(* Schneider Machine Expert - Basic project _M5.4 Schedule Block, file version 2.6.0.0 *)
(* CompanyInformations: Name=Schneider Electric, PhoneNumber=+44 870 608 8608, Street=Stafford Park 5, City=Telford, ZipCode=TF3 3BL, Country=United Kingdom, WebSite=se.com/uk *)
(* ProjectInformations: Name=Training M221, Description=Training of the Modicon M221.
We are going to work with a Conveyor belt machine.
During this trainignn we will add more features to this machine to understand how to use the software. *)
(* UserInformations: LastName=Ahumada, FirstName=Leandro, PhoneNumber=+44 870 608 8608, CellNumber=+44 870 608 8608, Email=gb-customerservices@schneider-electric.com, Street=Stafford Park 5, City=Telford, ZipCode=TF3 3BL, Country=United Kingdom *)

HARDWARE
  Cpu 0: TM221CE24R
  EthernetConfiguration: NetworkName=M221, IpAllocationMode=FixedAddress, IpAddress=192.168.1.221, SubnetMask=255.255.255.0
  SerialLineConfiguration: Baud=Baud19200, Parity=ParityEven, DataBits=DataBits8, StopBits=StopBits1, PhysicalMedium=PhysicalMediumRs485, TransmissionMode=TransmissionModeModbusRtu, SlaveId=1, Addressing=SlaveAddressing
  MastTask: UsePeriodScanMode=false, PeriodScan=100
  FastTask: Period=255
  CpuBehavior: StartingMode=StartAsPreviousState, AutoSaveRamOnEeprom=true, WatchdogPeriod=250

SYMBOLS  (address, symbol, comment, settings)
  %M0       AUX_MOTOR  "Auxiliar motor"
  %M1       AUX_MACHINE  "Auxiliar Machine"
  %M10      MI_START  "M Start pushbutton"
  %M11      MI_STOP  "M Stop pushbutton"
  %M12      MI_SENSOR  "M Photo-Electric sensor"
  %M20      CMD_COUNTER_RESET
  %M21      IND_COUNTER_REACHED
  %M22      CFG_SCH_MONDAY
  %M23      CFG_SCH_TUESDAY
  %M24      CFG_SCH_WEDNESDAY
  %M25      CFG_SCH_THURSDAY
  %M26      CFG_SCH_FRIDAY
  %M27      CFG_SCH_SATURDAY
  %M28      CFG_SCH_SUNDAY
  %M80      PET_RTC_ENABLE  "At state 1, the RD and WR input values are read continuously to determine the action to take."
  %M81      PET_RTC_READ  "RD = 1 and WR = 0. Read the RTC value."
  %M82      PET_RTC_WRITE  "RD = 0 and WR = 1. When the rising edge of WR is detected, update the RTC using the object values specified in the RTC parameter"
  %M83      IND_RTC_DONE  "Set to 1 when the RTC is successfully read from or written to."
  %M84      IND_RTC_ERROR  "The ErrorId output object indicates the cause of the error."
  %M90      IND_ALARM_SYSTEM
  %M100     PET_ACK
  %M101     ALARM_01
  %M102     ALARM_02
  %MW0      IND_MOTOR_COUNTER
  %MW1      IND_MOTOR_TIME
  %MW2      AUX_RTC_ACTUAL_TOTAL_MM
  %MW3      AUX_MACHINE_ON_TOTAL_MM
  %MW4      AUX_MACHINE_OFF_TOTAL_MM
  %MW10     CFG_TIMER_MOTOR
  %MW11     CFG_COUNTER_MOTOR
  %MW12     CFG_MACHINE_ON_HH
  %MW13     CFG_MACHINE_ON_MM
  %MW14     CFG_MACHINE_OFF_HH
  %MW15     CFG_MACHINE_OFF_MM
  %MW20     CFG_SCH_STARTDAY  "Config. - Schedule - Start day"
  %MW21     CFG_SCH_STARTMONTH  "Config. - Schedule - Start month"
  %MW22     CFG_SCH_STARTHOUR  "Config. - Schedule - Start hour"
  %MW23     CFG_SCH_STARTMIN  "Config. - Schedule - Start min"
  %MW24     CFG_SCH_ENDDAY  "Config. - Schedule - End day"
  %MW25     CFG_SCH_ENDMONTH  "Config. - Schedule - End month"
  %MW26     CFG_SCH_ENDHOUR  "Config. - Schedule - End hour"
  %MW27     CFG_SCH_ENDMIN
  %MW28     CFG_SCH_DOW  "Config. - Schedule - Day of week"
  %MW41     IND_RTC_IDERROR
  %MW42     IND_RTC_ACTUAL_DAY
  %MW43     IND_RTC_ACTUAL_MONTH
  %MW44     IND_RTC_ACTUAL_YEAR
  %MW45     IND_RTC_ACTUAL_HH
  %MW46     IND_RTC_ACTUAL_MM
  %MW47     IND_RTC_ACTUAL_SS
  %MW48     IND_RTC_ACTUAL_DAYOFWEEK
  %MW50     IND_RTC_WRITE_DAY
  %MW51     IND_RTC_WRITE_MONTH
  %MW52     IND_RTC_WRITE_YEAR
  %MW53     IND_RTC_WRITE_HH
  %MW54     IND_RTC_WRITE_MM
  %MW55     IND_RTC_WRITE_SS
  %MW100    VAR_A
  %MW101    VAR_B
  %MW102    VAR_C
  %MF104    VAR_D
  %TM0      TIMER_MOTOR_ON  [Preset=5, Base=OneSecond]
  %SCH0       [Configured=true, OutputBit=%M1, StartDate=2012-01-01T00:00:00, EndDate=2012-01-01T00:00:00]
  %RTC0     INST_RTC  [Day(Value(int=24)), Month(Value(int=12)), Year(Value(int=2019)), Hours(Value(int=0)), Minutes(Value(int=0)), Seconds(Value(int=0))]
  %I0.0     I_START  "Start pushbutton"
  %I0.1     I_STOP  "Stop pushbutton"
  %I0.5     I_SENSOR  "Photo-Electric sensor"
  %Q0.0     Q_MOTOR  "Motor"
  %Q0.1     Q_MACHINE_ON
  %Q0.2     Q_ALARM
  %Q0.3     Q_MACHINE_DISABLED

POU PRG_CONFIG
  (* SectionNumber=1 *)

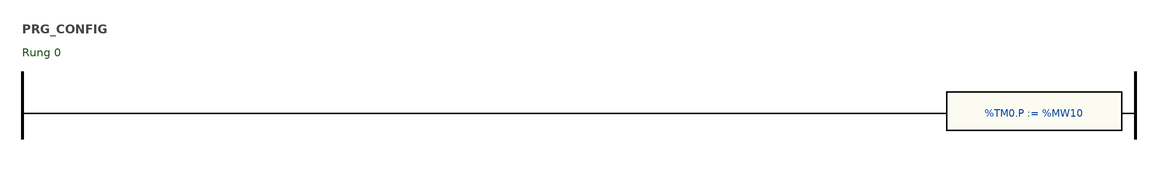

// Rung 0
  LD 1
  [ %TM0.P := %MW10 ]     (* TIMER_MOTOR_ON, CFG_TIMER_MOTOR *)
  // as ST:
  //   TIMER_MOTOR_ON.P := CFG_TIMER_MOTOR;

POU PRG_RTC
  (* SectionNumber=2 *)

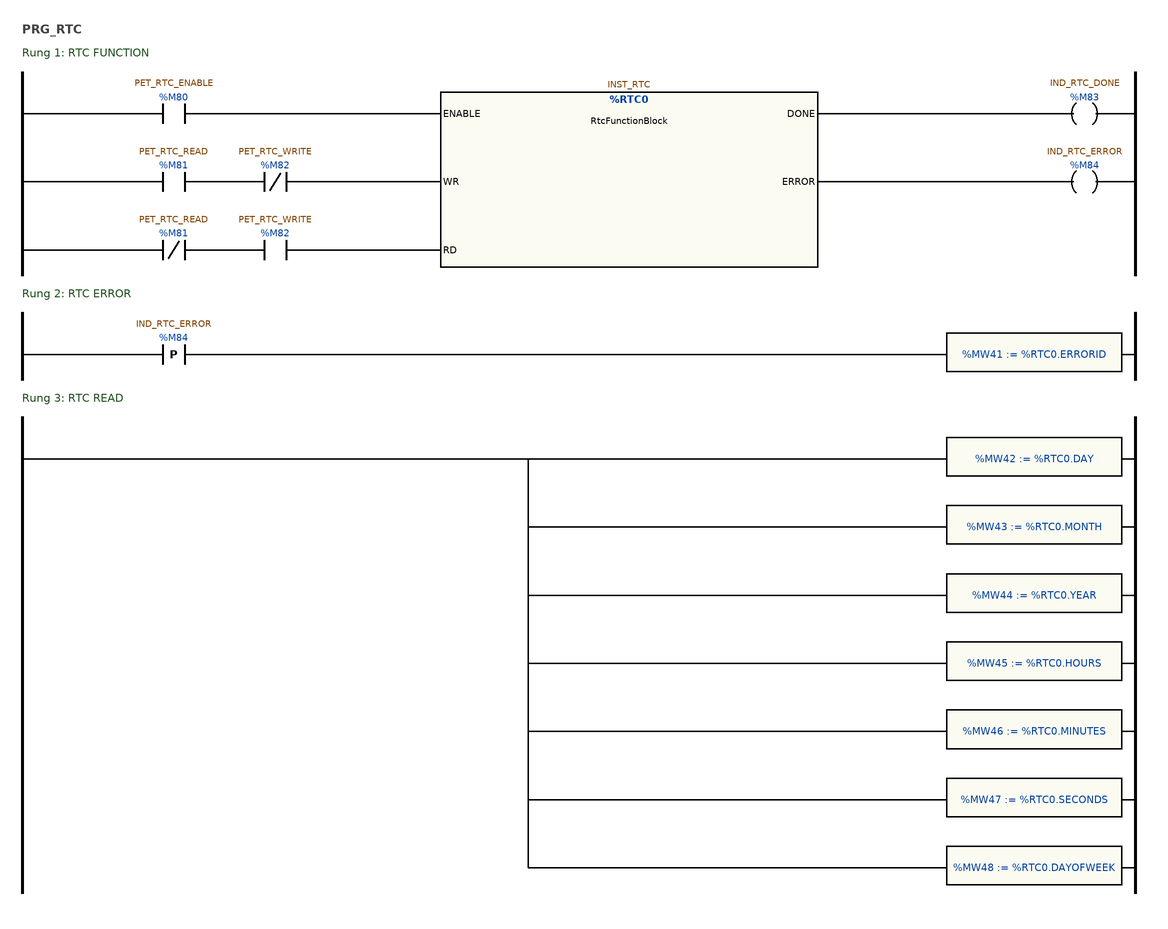

// Rung 1: RTC FUNCTION
  BLK %RTC0               (* INST_RTC *)
  LD %M80                 (* PET_RTC_ENABLE *)
  ENABLE
  LD %M81                 (* PET_RTC_READ *)
  ANDN %M82               (* PET_RTC_WRITE *)
  WR
  LDN %M81                (* PET_RTC_READ *)
  AND %M82                (* PET_RTC_WRITE *)
  RD
  OUT_BLK
  LD DONE
  ST %M83                 (* IND_RTC_DONE *)
  LD ERROR
  ST %M84                 (* IND_RTC_ERROR *)
  END_BLK
  // as ST:
  //   INST_RTC(ENABLE := PET_RTC_ENABLE, WR := PET_RTC_READ AND NOT PET_RTC_WRITE, RD := NOT PET_RTC_READ AND PET_RTC_WRITE);
  //   IND_RTC_DONE := INST_RTC.DONE;
  //   IND_RTC_ERROR := INST_RTC.ERROR;

// Rung 2: RTC ERROR
  LDR %M84                (* IND_RTC_ERROR *)
  [ %MW41 := %RTC0.ERRORID ](* IND_RTC_IDERROR, INST_RTC *)
  // as ST:
  //   IF RISING(IND_RTC_ERROR) THEN IND_RTC_IDERROR := INST_RTC.ERRORID; END_IF;

// Rung 3: RTC READ
  LD 1
  [ %MW42 := %RTC0.DAY ]  (* IND_RTC_ACTUAL_DAY, INST_RTC *)
  [ %MW43 := %RTC0.MONTH ](* IND_RTC_ACTUAL_MONTH, INST_RTC *)
  [ %MW44 := %RTC0.YEAR ] (* IND_RTC_ACTUAL_YEAR, INST_RTC *)
  [ %MW45 := %RTC0.HOURS ](* IND_RTC_ACTUAL_HH, INST_RTC *)
  [ %MW46 := %RTC0.MINUTES ](* IND_RTC_ACTUAL_MM, INST_RTC *)
  [ %MW47 := %RTC0.SECONDS ](* IND_RTC_ACTUAL_SS, INST_RTC *)
  [ %MW48 := %RTC0.DAYOFWEEK ](* IND_RTC_ACTUAL_DAYOFWEEK, INST_RTC *)
  // as ST:
  //   IND_RTC_ACTUAL_DAY := INST_RTC.DAY;
  //   IND_RTC_ACTUAL_MONTH := INST_RTC.MONTH;
  //   IND_RTC_ACTUAL_YEAR := INST_RTC.YEAR;
  //   IND_RTC_ACTUAL_HH := INST_RTC.HOURS;
  //   IND_RTC_ACTUAL_MM := INST_RTC.MINUTES;
  //   IND_RTC_ACTUAL_SS := INST_RTC.SECONDS;
  //   IND_RTC_ACTUAL_DAYOFWEEK := INST_RTC.DAYOFWEEK;

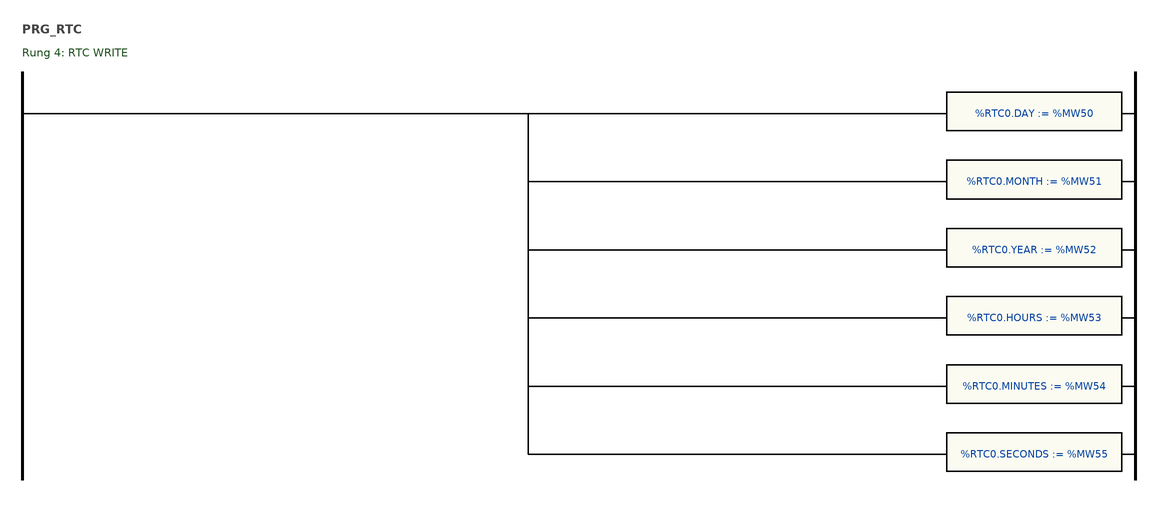

// Rung 4: RTC WRITE
  LD 1
  [ %RTC0.DAY := %MW50 ]  (* INST_RTC, IND_RTC_WRITE_DAY *)
  [ %RTC0.MONTH := %MW51 ](* INST_RTC, IND_RTC_WRITE_MONTH *)
  [ %RTC0.YEAR := %MW52 ] (* INST_RTC, IND_RTC_WRITE_YEAR *)
  [ %RTC0.HOURS := %MW53 ](* INST_RTC, IND_RTC_WRITE_HH *)
  [ %RTC0.MINUTES := %MW54 ](* INST_RTC, IND_RTC_WRITE_MM *)
  [ %RTC0.SECONDS := %MW55 ](* INST_RTC, IND_RTC_WRITE_SS *)
  // as ST:
  //   INST_RTC.DAY := IND_RTC_WRITE_DAY;
  //   INST_RTC.MONTH := IND_RTC_WRITE_MONTH;
  //   INST_RTC.YEAR := IND_RTC_WRITE_YEAR;
  //   INST_RTC.HOURS := IND_RTC_WRITE_HH;
  //   INST_RTC.MINUTES := IND_RTC_WRITE_MM;
  //   INST_RTC.SECONDS := IND_RTC_WRITE_SS;

POU PRG_SCHEDULE
  (* SectionNumber=3 *)

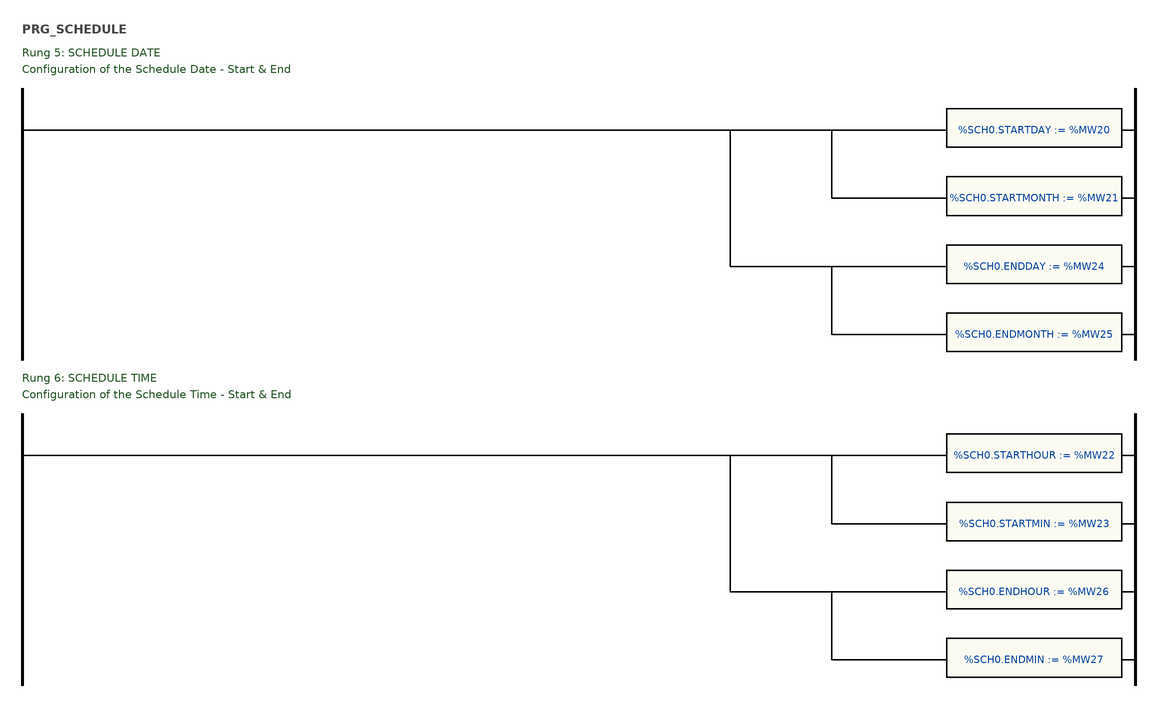

// Rung 5: SCHEDULE DATE
// Configuration of the Schedule Date - Start & End
  LD 1
  [ %SCH0.STARTDAY := %MW20 ](* CFG_SCH_STARTDAY *)
  [ %SCH0.STARTMONTH := %MW21 ](* CFG_SCH_STARTMONTH *)
  [ %SCH0.ENDDAY := %MW24 ](* CFG_SCH_ENDDAY *)
  [ %SCH0.ENDMONTH := %MW25 ](* CFG_SCH_ENDMONTH *)
  // as ST:
  //   %SCH0.STARTDAY := CFG_SCH_STARTDAY;
  //   %SCH0.STARTMONTH := CFG_SCH_STARTMONTH;
  //   %SCH0.ENDDAY := CFG_SCH_ENDDAY;
  //   %SCH0.ENDMONTH := CFG_SCH_ENDMONTH;

// Rung 6: SCHEDULE TIME
// Configuration of the Schedule Time - Start & End
  LD 1
  [ %SCH0.STARTHOUR := %MW22 ](* CFG_SCH_STARTHOUR *)
  [ %SCH0.STARTMIN := %MW23 ](* CFG_SCH_STARTMIN *)
  [ %SCH0.ENDHOUR := %MW26 ](* CFG_SCH_ENDHOUR *)
  [ %SCH0.ENDMIN := %MW27 ](* CFG_SCH_ENDMIN *)
  // as ST:
  //   %SCH0.STARTHOUR := CFG_SCH_STARTHOUR;
  //   %SCH0.STARTMIN := CFG_SCH_STARTMIN;
  //   %SCH0.ENDHOUR := CFG_SCH_ENDHOUR;
  //   %SCH0.ENDMIN := CFG_SCH_ENDMIN;

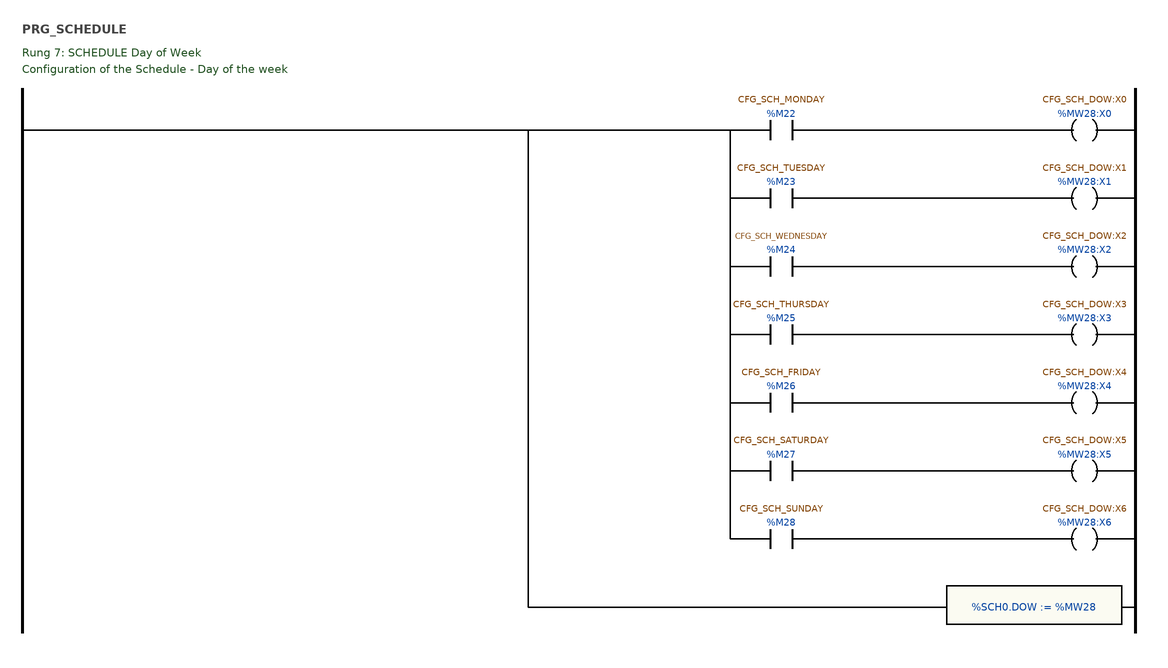

// Rung 7: SCHEDULE Day of Week
// Configuration of the Schedule - Day of the week
  LD 1
  MPS
  AND %M22                (* CFG_SCH_MONDAY *)
  ST %MW28:X0             (* CFG_SCH_DOW *)
  MRD
  AND %M23                (* CFG_SCH_TUESDAY *)
  ST %MW28:X1             (* CFG_SCH_DOW *)
  MRD
  AND %M24                (* CFG_SCH_WEDNESDAY *)
  ST %MW28:X2             (* CFG_SCH_DOW *)
  MRD
  AND %M25                (* CFG_SCH_THURSDAY *)
  ST %MW28:X3             (* CFG_SCH_DOW *)
  MRD
  AND %M26                (* CFG_SCH_FRIDAY *)
  ST %MW28:X4             (* CFG_SCH_DOW *)
  MRD
  AND %M27                (* CFG_SCH_SATURDAY *)
  ST %MW28:X5             (* CFG_SCH_DOW *)
  MRD
  AND %M28                (* CFG_SCH_SUNDAY *)
  ST %MW28:X6             (* CFG_SCH_DOW *)
  MPP
  [ %SCH0.DOW := %MW28 ]  (* CFG_SCH_DOW *)
  // as ST:
  //   CFG_SCH_DOW:X0 := CFG_SCH_MONDAY;
  //   CFG_SCH_DOW:X1 := CFG_SCH_TUESDAY;
  //   CFG_SCH_DOW:X2 := CFG_SCH_WEDNESDAY;
  //   CFG_SCH_DOW:X3 := CFG_SCH_THURSDAY;
  //   CFG_SCH_DOW:X4 := CFG_SCH_FRIDAY;
  //   CFG_SCH_DOW:X5 := CFG_SCH_SATURDAY;
  //   CFG_SCH_DOW:X6 := CFG_SCH_SUNDAY;
  //   %SCH0.DOW := CFG_SCH_DOW;

POU PRG_INPUTS
  (* SectionNumber=4 *)

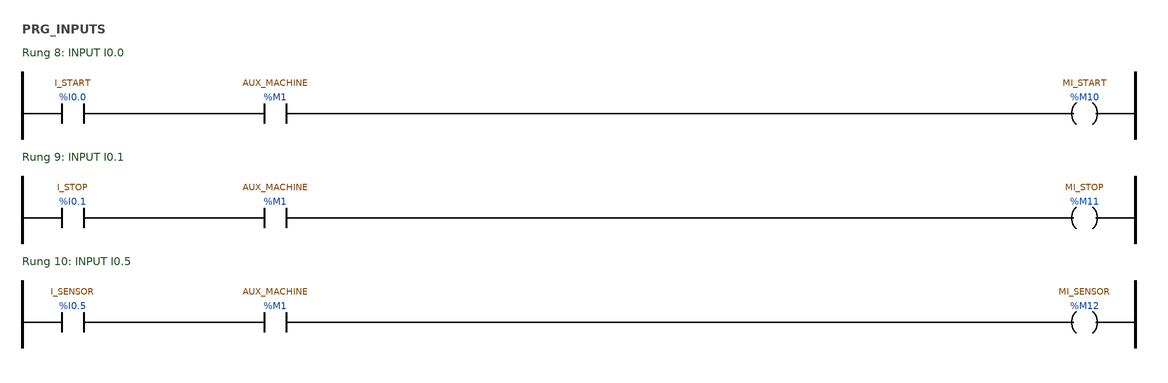

// Rung 8: INPUT I0.0
  LD %I0.0                (* I_START *)
  AND %M1                 (* AUX_MACHINE *)
  ST %M10                 (* MI_START *)
  // as ST:
  //   MI_START := I_START AND AUX_MACHINE;

// Rung 9: INPUT I0.1
  LD %I0.1                (* I_STOP *)
  AND %M1                 (* AUX_MACHINE *)
  ST %M11                 (* MI_STOP *)
  // as ST:
  //   MI_STOP := I_STOP AND AUX_MACHINE;

// Rung 10: INPUT I0.5
  LD %I0.5                (* I_SENSOR *)
  AND %M1                 (* AUX_MACHINE *)
  ST %M12                 (* MI_SENSOR *)
  // as ST:
  //   MI_SENSOR := I_SENSOR AND AUX_MACHINE;

POU PRG_MGMT
  (* SectionNumber=5 *)

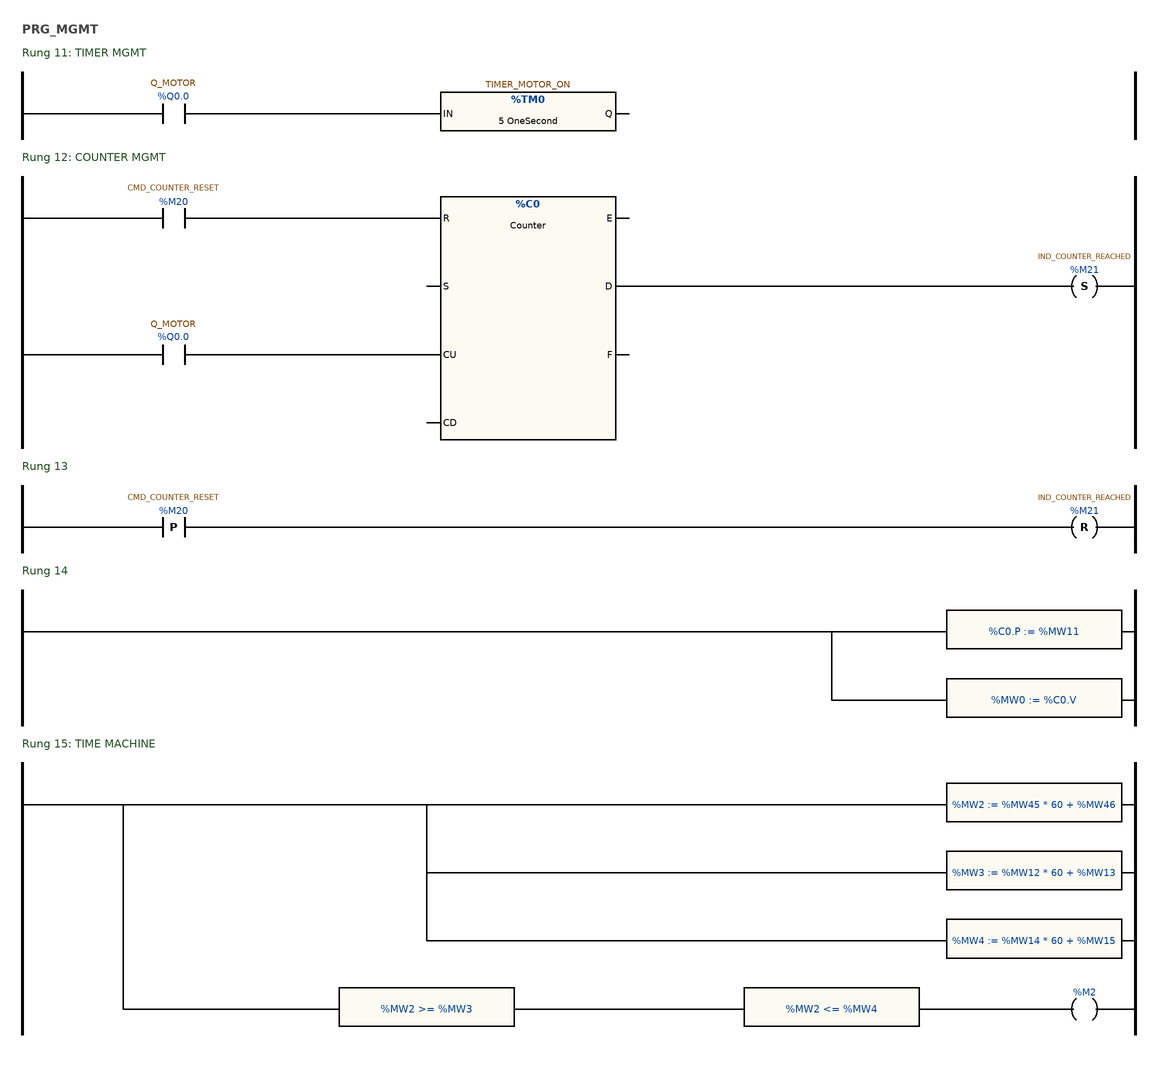

// Rung 11: TIMER MGMT
  BLK %TM0                (* TIMER_MOTOR_ON *)
  LD %Q0.0                (* Q_MOTOR *)
  IN
  END_BLK
  // as ST:
  //   TIMER_MOTOR_ON(IN := Q_MOTOR);

// Rung 12: COUNTER MGMT
  BLK %C0
  LD %M20                 (* CMD_COUNTER_RESET *)
  R
  LD %Q0.0                (* Q_MOTOR *)
  CU
  OUT_BLK
  LD D
  S %M21                  (* IND_COUNTER_REACHED *)
  END_BLK
  // as ST:
  //   %C0(R := CMD_COUNTER_RESET, CU := Q_MOTOR);
  //   IF %C0.D THEN IND_COUNTER_REACHED := TRUE; END_IF;

// Rung 13
  LDR %M20                (* CMD_COUNTER_RESET *)
  R %M21                  (* IND_COUNTER_REACHED *)
  // as ST:
  //   IF RISING(CMD_COUNTER_RESET) THEN IND_COUNTER_REACHED := FALSE; END_IF;

// Rung 14
  LD 1
  [ %C0.P := %MW11 ]      (* CFG_COUNTER_MOTOR *)
  [ %MW0 := %C0.V ]       (* IND_MOTOR_COUNTER *)
  // as ST:
  //   %C0.P := CFG_COUNTER_MOTOR;
  //   IND_MOTOR_COUNTER := %C0.V;

// Rung 15: TIME MACHINE
  LD 1
  MPS
  [ %MW2 := %MW45 * 60 + %MW46 ](* AUX_RTC_ACTUAL_TOTAL_MM, IND_RTC_ACTUAL_HH, IND_RTC_ACTUAL_MM *)
  MRD
  [ %MW3 := %MW12 * 60 + %MW13 ](* AUX_MACHINE_ON_TOTAL_MM, CFG_MACHINE_ON_HH, CFG_MACHINE_ON_MM *)
  MRD
  [ %MW4 := %MW14 * 60 + %MW15 ](* AUX_MACHINE_OFF_TOTAL_MM, CFG_MACHINE_OFF_HH, CFG_MACHINE_OFF_MM *)
  MPP
  AND [ %MW2 >= %MW3 ]    (* AUX_RTC_ACTUAL_TOTAL_MM, AUX_MACHINE_ON_TOTAL_MM *)
  AND [ %MW2 <= %MW4 ]    (* AUX_RTC_ACTUAL_TOTAL_MM, AUX_MACHINE_OFF_TOTAL_MM *)
  ST %M2
  // as ST:
  //   AUX_RTC_ACTUAL_TOTAL_MM := IND_RTC_ACTUAL_HH * 60 + IND_RTC_ACTUAL_MM;
  //   AUX_MACHINE_ON_TOTAL_MM := CFG_MACHINE_ON_HH * 60 + CFG_MACHINE_ON_MM;
  //   AUX_MACHINE_OFF_TOTAL_MM := CFG_MACHINE_OFF_HH * 60 + CFG_MACHINE_OFF_MM;
  //   %M2 := AUX_RTC_ACTUAL_TOTAL_MM >= AUX_MACHINE_ON_TOTAL_MM AND AUX_RTC_ACTUAL_TOTAL_MM <= AUX_MACHINE_OFF_TOTAL_MM;

POU PRG_ALARMS
  (* SectionNumber=6 *)

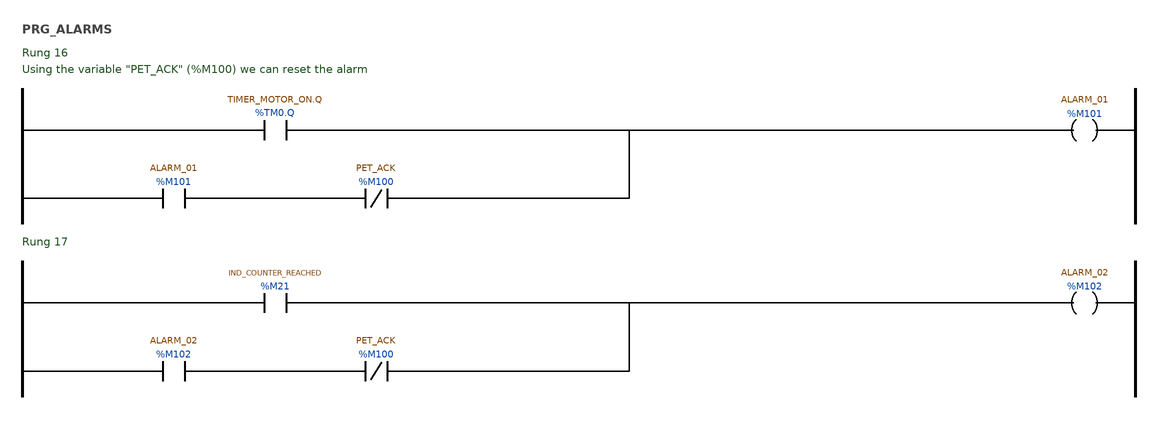

// Rung 16
// Using the variable "PET_ACK" (%M100) we can reset the alarm
  LD 1
  AND %TM0.Q              (* TIMER_MOTOR_ON *)
  OR( %M101               (* ALARM_01 *)
  ANDN %M100              (* PET_ACK *)
  )
  ST %M101                (* ALARM_01 *)
  // as ST:
  //   ALARM_01 := TIMER_MOTOR_ON.Q OR ALARM_01 AND NOT PET_ACK;

// Rung 17
  LD 1
  AND %M21                (* IND_COUNTER_REACHED *)
  OR( %M102               (* ALARM_02 *)
  ANDN %M100              (* PET_ACK *)
  )
  ST %M102                (* ALARM_02 *)
  // as ST:
  //   ALARM_02 := IND_COUNTER_REACHED OR ALARM_02 AND NOT PET_ACK;

POU PRG_GRAL_ALARMS
  (* SectionNumber=7 *)

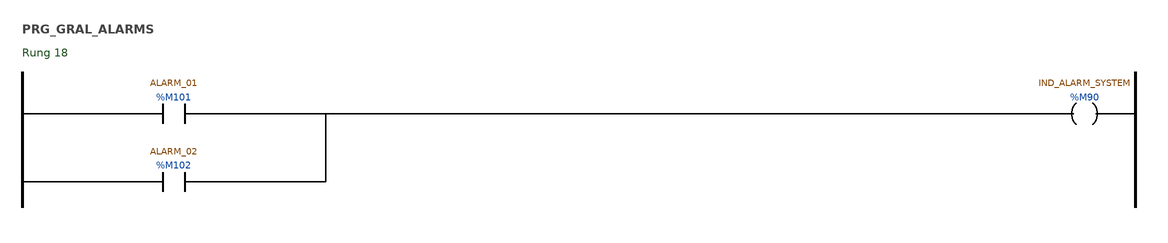

// Rung 18
  LD %M101                (* ALARM_01 *)
  OR %M102                (* ALARM_02 *)
  ST %M90                 (* IND_ALARM_SYSTEM *)
  // as ST:
  //   IND_ALARM_SYSTEM := ALARM_01 OR ALARM_02;

POU PRG_CONTROL
  (* SectionNumber=8 *)

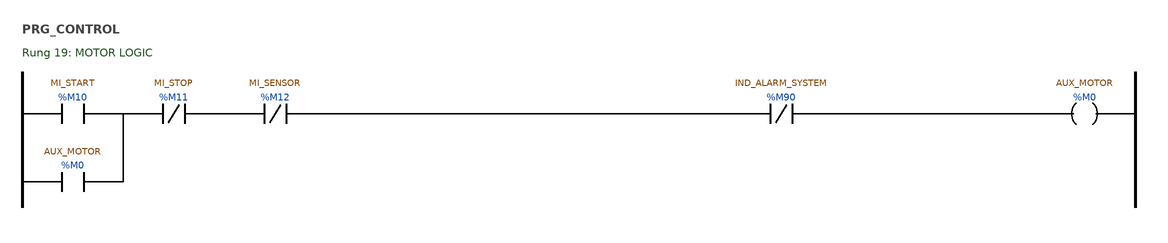

// Rung 19: MOTOR LOGIC
  LD %M10                 (* MI_START *)
  OR %M0                  (* AUX_MOTOR *)
  ANDN %M11               (* MI_STOP *)
  ANDN %M12               (* MI_SENSOR *)
  ANDN %M90               (* IND_ALARM_SYSTEM *)
  ST %M0                  (* AUX_MOTOR *)
  // as ST:
  //   AUX_MOTOR := (MI_START OR AUX_MOTOR) AND NOT MI_STOP AND NOT MI_SENSOR AND NOT IND_ALARM_SYSTEM;

POU PRG_OUTPUT
  (* SectionNumber=9 *)

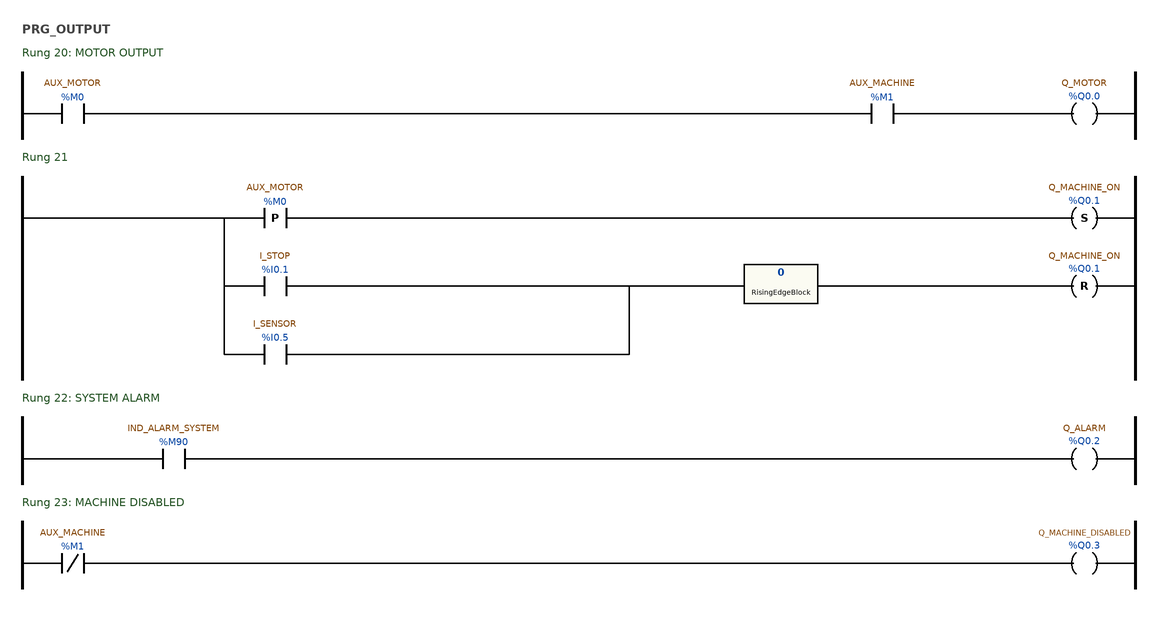

// Rung 20: MOTOR OUTPUT
  LD %M0                  (* AUX_MOTOR *)
  AND %M1                 (* AUX_MACHINE *)
  ST %Q0.0                (* Q_MOTOR *)
  // as ST:
  //   Q_MOTOR := AUX_MOTOR AND AUX_MACHINE;

// Rung 21
  LD 1
  MPS
  ANDR %M0                (* AUX_MOTOR *)
  S %Q0.1                 (* Q_MACHINE_ON *)
  MPP
  AND( %I0.1              (* I_STOP *)
  OR %I0.5                (* I_SENSOR *)
  )
  RISING0
  R %Q0.1                 (* Q_MACHINE_ON *)
  // as ST:
  //   IF RISING(AUX_MOTOR) THEN Q_MACHINE_ON := TRUE; END_IF;
  //   IF RISING(I_STOP OR I_SENSOR) THEN Q_MACHINE_ON := FALSE; END_IF;

// Rung 22: SYSTEM ALARM
  LD %M90                 (* IND_ALARM_SYSTEM *)
  ST %Q0.2                (* Q_ALARM *)
  // as ST:
  //   Q_ALARM := IND_ALARM_SYSTEM;

// Rung 23: MACHINE DISABLED
  LDN %M1                 (* AUX_MACHINE *)
  ST %Q0.3                (* Q_MACHINE_DISABLED *)
  // as ST:
  //   Q_MACHINE_DISABLED := NOT AUX_MACHINE;
